// TIA Portal project "Ventilacion_analoga_ejercisio_2" (V15)
// Trabajo Asignado Por el profesor Juan Guillermo

(* hardware
DEVICE "S7-1200 station_1"  S7-1200 Station
   slot 0: "Rack_0"  S7-1200 Rack  Rack  V1.0
   slot 1: "PLC_1"  CPU 1214C DC/DC/DC  6ES7 214-1AG40-0XB0  V4.2
   slot 2: "AI 4x13BIT_2"  6ES7 231-4HD32-0XB0  V2.0
*)

// ===== PLC "PLC_1"  CPU 1214C DC/DC/DC =====

VAR_GLOBAL   // PLC tag table "Tabla de variables estándar"
   "Entrada_Termocupla_4_20_mA" AT %IW112 : Word;
   "Tag_1" AT %MD20 : Real;
   "Temperatura_PLC" AT %MD24 : Real;
   "Inicio" AT %I0.0 : Bool;
   "Paro" AT %I0.1 : Bool;
   "Sistema_Activo" AT %M5.0 : Bool;
   "Ventilador_1" AT %Q0.0 : Bool;
   "Marca_alarma" AT %M5.1 : Bool;
   "Salida_Alarma_1" AT %Q0.1 : Bool;
END_VAR

// folder: System blocks/Program resources

DATA_BLOCK "T1"   // DB1
{ S7_Optimized_Access := 'TRUE' }
AUTHOR : Simatic
FAMILY : IEC
NAME : IEC_TMR
VERSION : 1.0
// stored: InstanceOfName IEC_TIMER
"IEC_TIMER"
BEGIN
END_DATA_BLOCK

DATA_BLOCK "T2"   // DB2
{ S7_Optimized_Access := 'TRUE' }
AUTHOR : Simatic
FAMILY : IEC
NAME : IEC_TMR
VERSION : 1.0
// stored: InstanceOfName IEC_TIMER
"IEC_TIMER"
BEGIN
END_DATA_BLOCK

// folder: (top level)

FUNCTION "Señales" : Void   // FC1, LAD
{ S7_Optimized_Access := 'TRUE' }
VERSION : 0.1
BEGIN

REGION Network 1
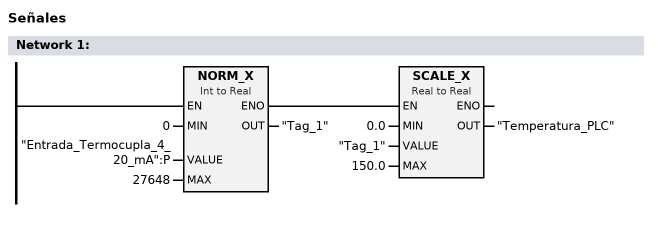
   RUNG wire#powerrail
      { S7_Templates := "[SrcType := Int, DestType := Real]" } Normalize(min := 0, value := "Entrada_Termocupla_4_20_mA":P, max := 27648, out => "Tag_1")
      { S7_Templates := "[SrcType := Real, DestType := Real]" } Scale(min := 0.0, value := "Tag_1", max := 150.0, out => "Temperatura_PLC")
   END_RUNG
   // the same network as SCL:
   "Tag_1" := NORM_X(MIN := 0, VALUE := "Entrada_Termocupla_4_20_mA":P, MAX := 27648);
   "Temperatura_PLC" := SCALE_X(MIN := 0.0, VALUE := "Tag_1", MAX := 150.0);
END_REGION
END_FUNCTION

FUNCTION "Enfriamiento" : Void   // FC2, LAD
{ S7_Optimized_Access := 'TRUE' }
VERSION : 0.1
   VAR_TEMP   // added for the SCL form of the ladder/FBD networks
      _w1 : Bool;
   END_VAR
BEGIN

REGION Network 1
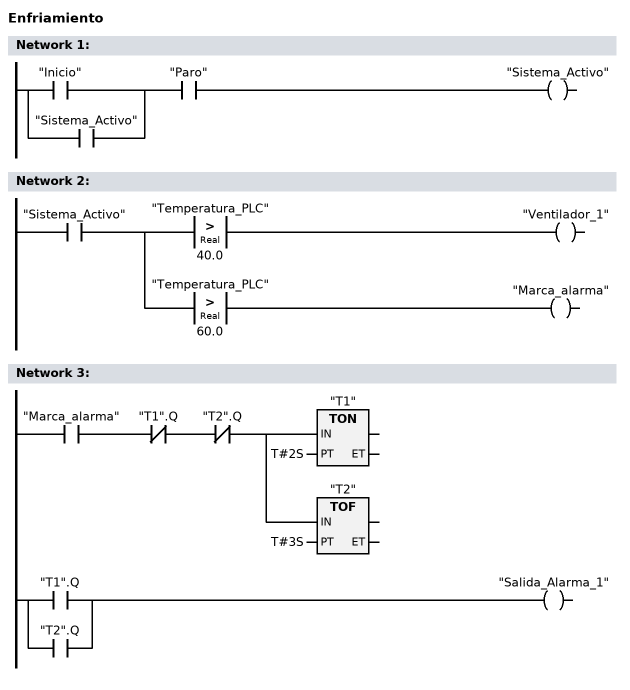
   RUNG wire#powerrail
      Contact( "Inicio" )
      wire#w1
      Contact( "Paro" )
      Coil( "Sistema_Activo" )
   END_RUNG
   RUNG wire#powerrail
      Contact( "Sistema_Activo" )
   END_RUNG wire#w1
   // the same network as SCL:
   "Sistema_Activo" := ("Inicio" OR "Sistema_Activo") AND "Paro";
END_REGION

REGION Network 2
   RUNG wire#powerrail
      Contact( "Sistema_Activo" )
      wire#w1
      { S7_Templates := "SrcType := Real" } GT_Contact(in1 := "Temperatura_PLC", in2 := 40.0)
      Coil( "Ventilador_1" )
   END_RUNG
   RUNG wire#w1
      { S7_Templates := "SrcType := Real" } GT_Contact(in1 := "Temperatura_PLC", in2 := 60.0)
      Coil( "Marca_alarma" )
   END_RUNG
   // the same network as SCL:
   "Ventilador_1" := "Sistema_Activo" AND ("Temperatura_PLC" > 40.0);
   "Marca_alarma" := "Sistema_Activo" AND ("Temperatura_PLC" > 60.0);
END_REGION

REGION Network 3
   #_w1 := "Marca_alarma" AND NOT "T1".Q AND NOT "T2".Q;
   "T1".TON(IN := #_w1, PT := T#2S);
   "T2".TOF(IN := #_w1, PT := T#3S);
   "Salida_Alarma_1" := "T1".Q OR "T2".Q;
END_REGION
END_FUNCTION

ORGANIZATION_BLOCK "Main"   // OB1, LAD, ProgramCycle
TITLE = "Main Program Sweep (Cycle)"
{ S7_Optimized_Access := 'TRUE' }
VERSION : 0.1
   VAR_INPUT
      Initial_Call : Bool;   // Initial call of this OB
      Remanence : Bool;   // =True, if remanent data are available
   END_VAR
BEGIN

REGION Network 1
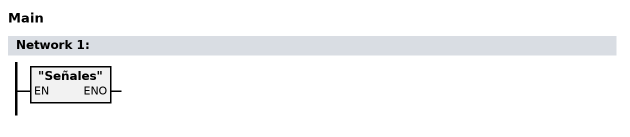
   RUNG wire#powerrail
      "Señales"()
   END_RUNG
   // the same network as SCL:
   "Señales"();
END_REGION
END_ORGANIZATION_BLOCK